// TwinCAT 3 PLC project _1Calcul
// ProgramVersion: 3.1.4020.2
// libraries:
//   Tc2_Standard, * (Beckhoff Automation GmbH)
//   Tc2_System, * (Beckhoff Automation GmbH)
//   Tc3_Module, * (Beckhoff Automation GmbH)
// project tree:
//   / PlcTask.TcTTO
//   POUs/ f_calcul.TcPOU, MAIN.TcPOU
// real-time tasks:
//   TASK PlcTask: cycle T#1ms, priority 20, ADS port 350
// I/O:
//   DEVICE Gerät 2 (EtherCAT)
//     Box 1 (BK1150)
// variable links:
//   GestionDesModesDeMarche/GestionDesModesDeMarche Instance <-> Device 2 (EtherCAT)/Box 1 (BK1150)
//     PlcTask Inputs/GVL.fbAct1.IxSensIn <-> Term 6 (KL1408)/Channel 2/Eingang
//     PlcTask Inputs/GVL.fbAct2.IxSensIn <-> Term 6 (KL1408)/Channel 4/Eingang
//     PlcTask Inputs/GVL.fbAct1.IxSensOut <-> Term 6 (KL1408)/Channel 1/Eingang
//     PlcTask Inputs/GVL.fbAct2.IxSensOut <-> Term 6 (KL1408)/Channel 3/Eingang
//     PlcTask Inputs/GVL.fbAct3.IxSensOut <-> Term 6 (KL1408)/Channel 5/Eingang
//     PlcTask Inputs/GVL.fbAct1.xReset <-> Term 6 (KL1408)/Channel 8/Eingang
//     PlcTask Inputs/GVL.fbAct2.xReset <-> Term 6 (KL1408)/Channel 8/Eingang
//     PlcTask Inputs/GVL.fbAct3.xReset <-> Term 6 (KL1408)/Channel 8/Eingang
//     PlcTask Inputs/GVL.stIO.stIn.IxAruIO <-> Term 7 (KL1408)/Channel 1/Eingang
//     PlcTask Inputs/GVL.stIO.stIn.xAuto <-> Term 7 (KL1408)/Channel 3/Eingang
//     PlcTask Inputs/GVL.stIO.stIn.xManual <-> Term 7 (KL1408)/Channel 2/Eingang
//     PlcTask Inputs/GVL.stIO.stIn.xResetIO <-> Term 6 (KL1408)/Channel 8/Eingang
//     PlcTask Inputs/GVL.stIO.stIn.xStartIO <-> Term 6 (KL1408)/Channel 6/Eingang
//     PlcTask Inputs/GVL.stIO.stIn.xStopIO <-> Term 6 (KL1408)/Channel 7/Eingang
//     PlcTask Outputs/GVL.fbAct1.QxInOutput <-> Term 8 (KL2408)/Channel 6/Ausgang
//     PlcTask Outputs/GVL.fbAct2.QxInOutput <-> Term 8 (KL2408)/Channel 8/Ausgang
//     PlcTask Outputs/GVL.fbAct1.QxOutOutput <-> Term 8 (KL2408)/Channel 5/Ausgang
//     PlcTask Outputs/GVL.fbAct2.QxOutOutput <-> Term 8 (KL2408)/Channel 7/Ausgang
//     PlcTask Outputs/GVL.fbAct3.QxOutOutput <-> Term 9 (KL2408)/Channel 1/Ausgang
//     PlcTask Outputs/GVL.fbAct1.QxVanneDeBloquage <-> Term 9 (KL2408)/Channel 2/Ausgang
//     PlcTask Outputs/GVL.stIO.stOut.QxLampeOrange <-> Term 8 (KL2408)/Channel 2/Ausgang
//     PlcTask Outputs/GVL.stIO.stOut.QxLampeRouge <-> Term 8 (KL2408)/Channel 1/Ausgang
//     PlcTask Outputs/GVL.stIO.stOut.QxLampeVerte <-> Term 8 (KL2408)/Channel 3/Ausgang

CONFIGURATION _1Calcul
    RESOURCE PLC ON TwinCAT3
        TASK PlcTask(INTERVAL := T#1ms, PRIORITY := 20);
        PROGRAM MAIN WITH PlcTask : MAIN;
    END_RESOURCE
END_CONFIGURATION

// ---- POUs/MAIN.TcPOU
PROGRAM MAIN
VAR
	MrAnglef: REAL;
	MrHypotenusef: REAL;
	MrResultat: REAL;
END_VAR

MrResultat:=f_calcul(MrAnglef,MrHypotenusef);

END_PROGRAM

// ---- POUs/f_calcul.TcPOU
FUNCTION f_calcul : REAL
VAR_INPUT
	IrAngle : REAL;
	IrHypotenuse : REAL;
END_VAR

f_calcul:=IrHypotenuse*SIN(IrAngle);

END_FUNCTION
